// TIA Portal project "Bai 4" (V16)

(* hardware
DEVICE "S7-1200 station_1"  S7-1200 Station
   slot 0: "Rack_0"  S7-1200 Rack  Rack  V1.0
   slot 1: "PLC_1"  CPU 1214C DC/DC/DC  6ES7 214-1AG40-0XB0  V4.1
   slot 2: "DQ 16xRelay_1"  SM 1222 DQ16 x relay  6ES7 222-1HH32-0XB0  V2.0
   slot 3: "AQ 1x12BIT_1"  AQ1 signal board  6ES7 232-4HA30-0XB0  V1.0
*)

// ===== PLC "PLC_1"  CPU 1214C DC/DC/DC =====

VAR_GLOBAL   // PLC tag table "Default tag table"
   "LQ1" AT %I0.2 : Bool;
   "LQ2" AT %I0.3 : Bool;
   "SQ1" AT %I0.4 : Bool;
   "SQ2" AT %I0.5 : Bool;
   "YV1" AT %Q9.1 : Bool;
   "YV2" AT %Q9.2 : Bool;
   "YV3" AT %Q9.3 : Bool;
   "YV4" AT %Q9.4 : Bool;
   "YV5" AT %Q9.5 : Bool;
   "YV6" AT %Q9.6 : Bool;
   "SQ3" AT %I0.6 : Bool;
   "Start" AT %I0.0 : Bool;
   "Stop" AT %I0.1 : Bool;
   "Ngat YV1" AT %M0.1 : Bool;
   "Giu Timer 1" AT %M0.0 : Bool;
   "Day YV2-4 ve" AT %M0.2 : Bool;
   "Bien hut" AT %M0.3 : Bool;
   "Ngat hut" AT %M0.4 : Bool;
   "Bien phu dieu khien Stop" AT %M0.6 : Bool;
   "Tat chuong trinh" AT %M1.0 : Bool;
END_VAR

// folder: System blocks/Program resources

DATA_BLOCK "T1"   // DB1
{ S7_Optimized_Access := 'TRUE' }
AUTHOR : Simatic
FAMILY : IEC
NAME : IEC_TMR
VERSION : 1.0
// stored: InstanceOfName IEC_TIMER
"IEC_TIMER"
BEGIN
END_DATA_BLOCK

DATA_BLOCK "T2"   // DB2
{ S7_Optimized_Access := 'TRUE' }
AUTHOR : Simatic
FAMILY : IEC
NAME : IEC_TMR
VERSION : 1.0
// stored: InstanceOfName IEC_TIMER
"IEC_TIMER"
BEGIN
END_DATA_BLOCK

// folder: (top level)

ORGANIZATION_BLOCK "Main"   // OB1, LAD, ProgramCycle
TITLE = "Main Program Sweep (Cycle)"
{ S7_Optimized_Access := 'TRUE' }
VERSION : 0.1
   VAR_INPUT
      Initial_Call : Bool;   // Initial call of this OB
      Remanence : Bool;   // =True, if remanent data are available
   END_VAR
   VAR_TEMP   // added for the SCL form of the ladder/FBD networks
      _w1 : Bool;
   END_VAR
BEGIN

REGION Network 1
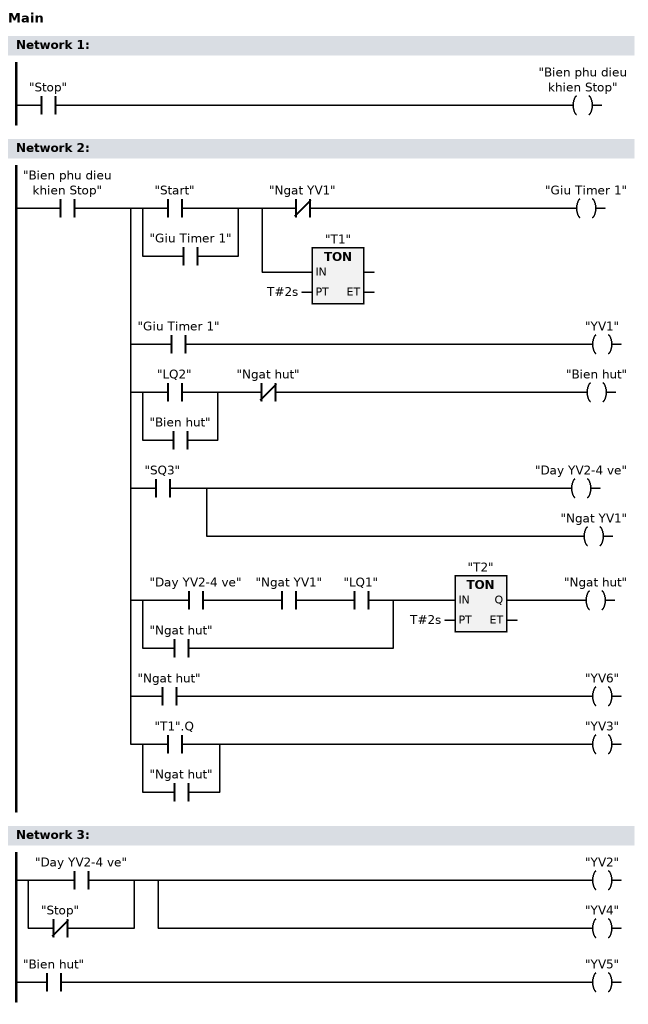
   RUNG wire#powerrail
      Contact( "Stop" )
      Coil( "Bien phu dieu khien Stop" )
   END_RUNG
   // the same network as SCL:
   "Bien phu dieu khien Stop" := "Stop";
END_REGION

REGION Network 2
   #_w1 := "Bien phu dieu khien Stop" AND ("Start" OR "Giu Timer 1");
   "Giu Timer 1" := #_w1 AND NOT "Ngat YV1";
   "T1".TON(IN := #_w1, PT := T#2s);
   "YV1" := "Bien phu dieu khien Stop" AND "Giu Timer 1";
   "Bien hut" := "Bien phu dieu khien Stop" AND ("LQ2" OR "Bien hut") AND NOT "Ngat hut";
   "Day YV2-4 ve" := "Bien phu dieu khien Stop" AND "SQ3";
   "Ngat YV1" := "Day YV2-4 ve";
   "T2".TON(IN := "Bien phu dieu khien Stop" AND (("Day YV2-4 ve" AND "Ngat YV1" AND "LQ1") OR "Ngat hut"),
            PT := T#2s);
   "Ngat hut" := "T2".Q;
   "YV6" := "Bien phu dieu khien Stop" AND "Ngat hut";
   "YV3" := "Bien phu dieu khien Stop" AND ("T1".Q OR "Ngat hut");
END_REGION

REGION Network 3
   RUNG wire#powerrail
      Contact( "Day YV2-4 ve" )
      wire#w1
      Coil( "YV2" )
   END_RUNG
   RUNG wire#powerrail
      I_Contact( "Stop" )
   END_RUNG wire#w1
   RUNG wire#w1
      Coil( "YV4" )
   END_RUNG
   RUNG wire#powerrail
      Contact( "Bien hut" )
      Coil( "YV5" )
   END_RUNG
   // the same network as SCL:
   "YV2" := "Day YV2-4 ve" OR NOT "Stop";
   "YV4" := "YV2";
   "YV5" := "Bien hut";
END_REGION
END_ORGANIZATION_BLOCK